// TIA Portal V20 export
TYPE "LWONIK_typeToSafetyLampStatus"
// stored: Access Published
   STRUCT
      HomeLampStatus : Bool;
      LampStatus1 : Bool;
      LampStatus2 : Bool;
      LampStatus3 : Bool;
      LampStatus4 : Bool;
      LampStatus5 : Bool;
      LampStatus6 : Bool;
   END_STRUCT;
END_TYPE
